// Mitsubishi GX Works2 project: part2   PLC: FX3G

// global labels: Global1
VAR_GLOBAL
  conveyor AT X007 : BOOL;
  conveyorLamp AT Y007 : BOOL;
  conveyorOff AT X001 : BOOL;
  magnet AT X002 : BOOL;
  magnetLamp AT Y002 : BOOL;
  vacume AT X003 : BOOL;
  vacumeLamp AT Y003 : BOOL;
  closeDoor AT X000 : BOOL;
  shreddLamp AT Y001 : BOOL;
  above4meter AT X004 : BOOL;
END_VAR
VAR_GLOBAL CONSTANT
  tenSec : INT := 100;
END_VAR
VAR_GLOBAL
  timer AT TC1 : BOOL;
  timerFinish AT TS1 : BOOL;
  above50 AT X005 : BOOL;
  above70 AT X006 : BOOL;
  washLamp AT Y010 : BOOL;
  vacumeLampp AT Y003 : BOOL;
  doorClose AT Y011 : BOOL;
  shreddLampp AT Y001 : BOOL;
  nisayon AT Y005 : BOOL;
  Timer1 AT TC1 : BOOL;
END_VAR
VAR_GLOBAL CONSTANT
  tenSecond : INT := 100;
END_VAR
VAR_GLOBAL
  shreddFinish AT Y005 : BOOL;
  Timer0 AT TC0 : BOOL;
END_VAR
VAR_GLOBAL CONSTANT
  countFour : INT := 70;
  countSeven : INT := 70;
END_VAR
VAR_GLOBAL
  switch4 AT Y004 : BOOL;
  Timer2 AT TC2 : BOOL;
END_VAR
VAR_GLOBAL CONSTANT
  countHalfSec : INT := 5;
END_VAR
VAR_GLOBAL
  Timer3 AT TS2 : BOOL;
  startFlickering AT M100 : BOOL;
  finished_sevenSec_timer AT TS0 : BOOL;
END_VAR
VAR_GLOBAL CONSTANT
  countSec : INT := 10;
END_VAR
VAR_GLOBAL
  Timer4 AT TC4 : BOOL;
  Timer5 AT TS4 : BOOL;
  switch11 AT M200 : BOOL;
  chen AT Y006 : BOOL;
  switch20 AT M60 : BOOL;
END_VAR

// task Task_01 (event TRUE, interval 0, priority 31): POU_01

PROGRAM POU_01
(* structured ladder/FBD written out as ST: instructions are called as NAME(EN, inputs, outputs); _pN, _eN, _tN stand for wires *)
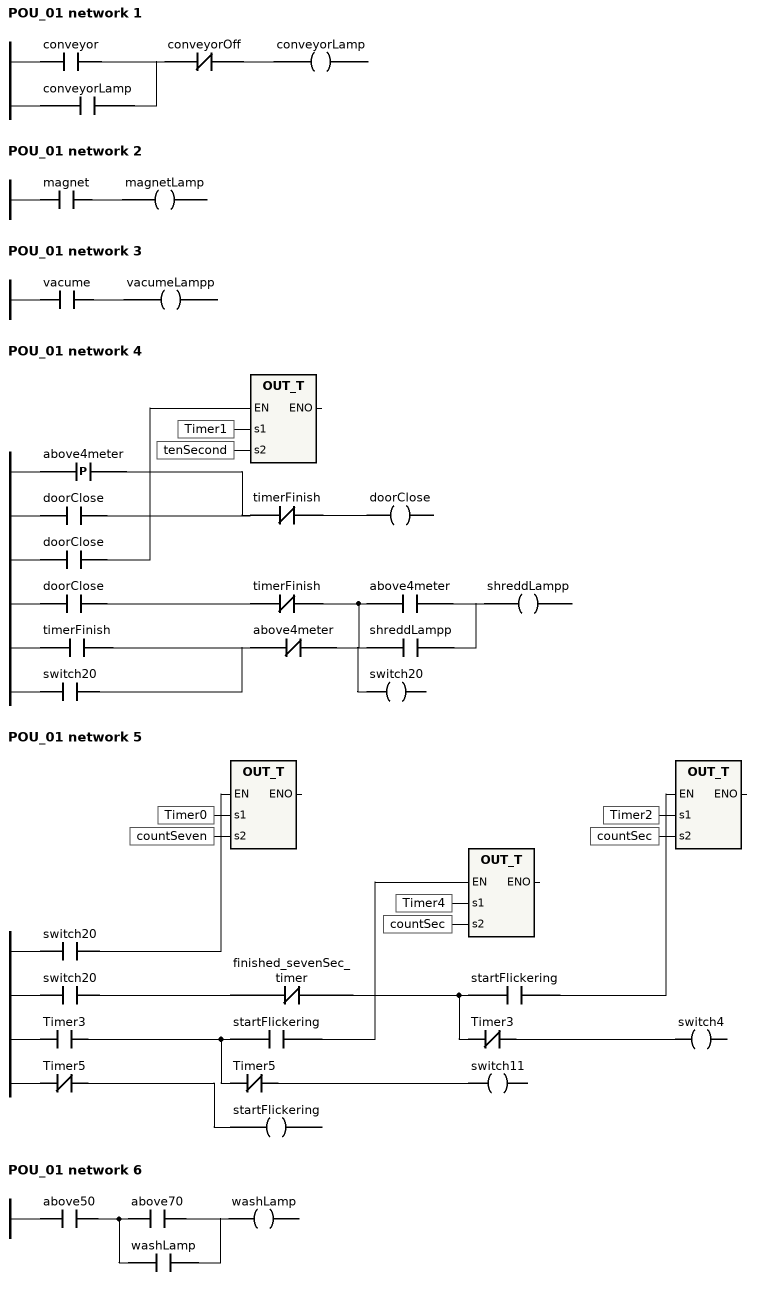
(* network 1 *)
conveyorLamp := (conveyor OR conveyorLamp) AND NOT conveyorOff;
(* network 2 *)
magnetLamp := magnet;
(* network 3 *)
vacumeLampp := vacume;
(* network 4 *)
doorClose := (LDP(TRUE, above4meter) OR doorClose) AND NOT timerFinish;
OUT_T(doorClose, Timer1, tenSecond);
_p1 := doorClose AND NOT timerFinish;
shreddLampp := (_p1 AND above4meter) OR (_p1 AND shreddLampp);
switch20 := (timerFinish OR switch20) AND NOT above4meter;
(* network 5 *)
OUT_T(switch20, Timer0, countSeven);
_p1 := switch20 AND NOT finished_sevenSec_timer;
OUT_T(_p1 AND startFlickering, Timer2, countSec);
switch4 := _p1 AND NOT Timer3;
OUT_T(Timer3 AND startFlickering, Timer4, countSec);
switch11 := Timer3 AND NOT Timer5;
startFlickering := NOT Timer5;
(* network 6 *)
washLamp := (above50 AND above70) OR (above50 AND washLamp);
END_PROGRAM
